TEXTLIST TextList_05
   = ''
END_TEXTLIST

(* stored: Version 1.1.0.1
   TextList TextList_05: Id {94a5d82e-a875-0f3c-0a7d-3fd2eba6c332} *)
